FUNCTION_BLOCK Robot_Update
VAR_INPUT
END_VAR
VAR_OUTPUT
	Free : BOOL;
	Error : Robot_Error;
END_VAR
VAR_IN_OUT
	Robot : UR3e_Robot;
END_VAR
VAR
	bitArray : BitStruct_Byte;
END_VAR

Error := Robot_Chek_errors(Robot:= Robot);

// chek of robot bezig is
IF (Robot.GPR_BIT[0] AND 2#00000001) = 2#00000001 THEN
	// zet run varibel FALSE zo dat robot de job niet bleift heralen
	bitArray.Value := Robot.GPR1[0];
	bitArray.SValue.Bit0 := FALSE;
	Robot.GPR1[0] := bitArray.Value;
	Free := FALSE;
ELSE
	Free := TRUE;
END_IF

END_FUNCTION_BLOCK

(* stored: Version 1.1.0.1, ProductVersion 3.1.4024.10
   POU Robot_Update: Id {b5d7f035-0ac8-48b6-b8af-7218a9f22efd}, SpecialFunc None *)
